// TIA Portal V19 export
FUNCTION "FC10_AnalogInput" : Void   // FC10, LAD
TITLE = Analog Input
{ S7_Optimized_Access := 'TRUE' }
// stored: AutoNumber false, IsIECCheckEnabled true, SetENOAutomatically false
BEGIN

REGION Network 1: Convert input analog value in distance value
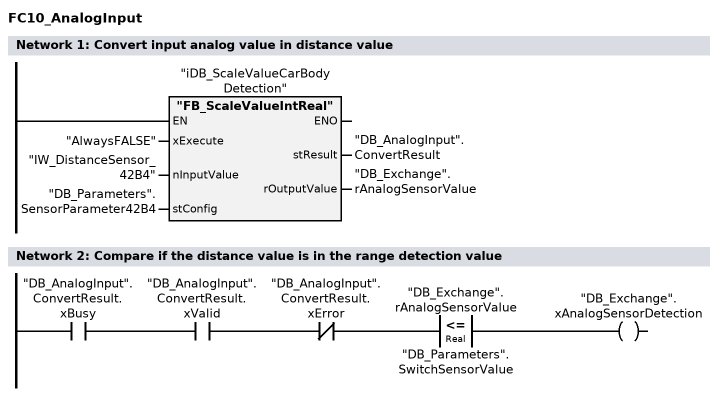
   RUNG wire#powerrail
      "iDB_ScaleValueCarBodyDetection"(xExecute := "AlwaysFALSE", nInputValue := "IW_DistanceSensor_42B4", stConfig := "DB_Parameters".SensorParameter42B4, stResult => "DB_AnalogInput".ConvertResult, rOutputValue => "DB_Exchange".rAnalogSensorValue)
   END_RUNG
   // the same network as SCL:
   "iDB_ScaleValueCarBodyDetection"(xExecute := "AlwaysFALSE",   // "FB_ScaleValueIntReal"
                           nInputValue := "IW_DistanceSensor_42B4",
                           stConfig := "DB_Parameters".SensorParameter42B4,
                           stResult => "DB_AnalogInput".ConvertResult,
                           rOutputValue => "DB_Exchange".rAnalogSensorValue);
END_REGION

REGION Network 2: Compare if the distance value is in the range detection value
   RUNG wire#powerrail
      Contact( "DB_AnalogInput".ConvertResult.xBusy )
      Contact( "DB_AnalogInput".ConvertResult.xValid )
      I_Contact( "DB_AnalogInput".ConvertResult.xError )
      { S7_Templates := "SrcType := Real" } LE_Contact(in1 := "DB_Exchange".rAnalogSensorValue, in2 := "DB_Parameters".SwitchSensorValue)
      Coil( "DB_Exchange".xAnalogSensorDetection )
   END_RUNG
   // the same network as SCL:
   "DB_Exchange".xAnalogSensorDetection := "DB_AnalogInput".ConvertResult.xBusy AND "DB_AnalogInput".ConvertResult.xValid AND NOT "DB_AnalogInput".ConvertResult.xError AND ("DB_Exchange".rAnalogSensorValue <= "DB_Parameters".SwitchSensorValue);
END_REGION
END_FUNCTION
